Yaskawa INFORM job: pointsmerc3.JBI

/JOB
//NAME pointsmerc3
//POS
///NPOS 0,0,0,0,0,0
///TOOL 1
///POSTYPE ROBOT
///RECTAN
///RCONF 1,0,0,0,0,0,0,0,0,0,0,0,0,0,0,0,0,0,0,0,0,0,0,0
//INST
///DATE 2021/02/10 13:51
///COMM
///ATTR SC,RW,RJ
////FRAME USER 2
///GROUP1 RB1
NOP
CALL JOB:DEBUT
'Part trajectory number: 0
CALL JOB:pointsmerc3TRJ0
'Part trajectory number: 1
CALL JOB:pointsmerc3TRJ1
'Part trajectory number: 2
CALL JOB:pointsmerc3TRJ2
CALL JOB:FIN
END
